// TwinCAT 3 PLC project Mcc
// ProgramVersion: 3.1.4024.0
// libraries:
//   Tc2_Standard, * (Beckhoff Automation GmbH)
//   Tc2_System, * (Beckhoff Automation GmbH)
//   Tc3_Module, * (Beckhoff Automation GmbH)
// project tree:
//   DUTs/ ST_WorkTime.TcDUT
//   POUs/Devices/ Button_NO.TcPOU, Label.TcPOU, Led.TcPOU, MccMotor.TcPOU, MotorContactor.TcPOU, MotorTermFuse.TcPOU, TaurusLed.TcPOU, WorkCounter.TcPOU
//   POUs/Devices/ITFs/ I_Button.TcIO, I_Label.TcIO, I_TaurusLed.TcIO, I_TermFuse.TcIO
//   POUs/ MAIN.TcPOU
// real-time tasks:
//   TASK PlcTask2: cycle T#10ms, priority 22, ADS port 352
// I/O:
//   DEVICE Device 1 (EtherCAT), AmsNetId 192.168.0.130.2.1
//     Term 1 (EK1200) [EK1200-5000 EtherCAT Power supply (2A E-Bus)]
//       Term 2 (EL2008) [EL2008 8Ch. Dig. Output 24V, 0.5A]
//       Term 3 (EL6022) [EL6022 Interface 2Ch. (RS422/485)]
//       Term 4 (EL9011) [EL9011 End Terminal]
//   DEVICE Device 3 (NOV-DP-RAM)
// variable links:
//   MotorControl Instance <-> Device 1 (EtherCAT)/Term 1 (EK1200)/Term 10 (EL2008)
//     PlcTask Outputs/Fermentation_001.MccRev_001.bContactor <-> Channel 1/Fermentation_001.MccRev_001.bContactor
//     PlcTask Outputs/Fermentation_001.MccRev_002.bContactor <-> Channel 2/Fermentation_001.MccRev_002.bContactor
//     PlcTask Outputs/Fermentation_001.MccRev_003.bContactor <-> Channel 3/Fermentation_001.MccRev_003.bContactor
//     PlcTask Outputs/Fermentation_001.MccRev_004.bContactor <-> Channel 4/Fermentation_001.MccRev_004.bContactor
//     PlcTask Outputs/Fermentation_001.MccRev_005.bContactor <-> Channel 5/Fermentation_001.MccRev_005.bContactor
//     PlcTask Outputs/Fermentation_001.MccRev_006.bContactor <-> Channel 6/Fermentation_001.MccRev_006.bContactor
//     PlcTask Outputs/Fermentation_001.MccRev_007.bContactor <-> Channel 7/Fermentation_001.MccRev_007.bContactor
//     PlcTask Outputs/Fermentation_001.MccRev_008.bContactor <-> Channel 8/Fermentation_001.MccRev_008.bContactor
//   MotorControl Instance <-> Device 1 (EtherCAT)/Term 1 (EK1200)/Term 11 (EL2008)
//     PlcTask Outputs/Fermentation_001.MccRev_009.bContactor <-> Channel 1/Fermentation_001.MccRev_009.bContactor
//     PlcTask Outputs/Fermentation_001.MccRev_010.bContactor <-> Channel 2/Fermentation_001.MccRev_010.bContactor
//     PlcTask Outputs/Fermentation_001.MccRev_011.bContactor <-> Channel 3/Fermentation_001.MccRev_011.bContactor
//     PlcTask Outputs/Fermentation_001.MccRev_012.bContactor <-> Channel 4/Fermentation_001.MccRev_012.bContactor
//     PlcTask Outputs/Fermentation_001.MccRev_013.bContactor <-> Channel 5/Fermentation_001.MccRev_013.bContactor
//     PlcTask Outputs/Fermentation_001.MccRev_014.bContactor <-> Channel 6/Fermentation_001.MccRev_014.bContactor
//     PlcTask Outputs/Fermentation_001.MccRev_015.bContactor <-> Channel 7/Fermentation_001.MccRev_015.bContactor
//     PlcTask Outputs/Fermentation_001.MccRev_016.bContactor <-> Channel 8/Fermentation_001.MccRev_016.bContactor
//   MotorControl Instance <-> Device 1 (EtherCAT)/Term 1 (EK1200)/Term 14 (EL3058)
//     PlcTask Inputs/Fermentation_001.TempSens_001.rRawTempValue <-> AI Standard Channel 1/Fermentation_001.TempSens_001.rRawTempValue
//   MotorControl Instance <-> Device 1 (EtherCAT)/Term 1 (EK1200)/Term 2 (EL2008)
//     PlcTask Outputs/Fermentation_001.MccRev_017.bContactor <-> Channel 1/Fermentation_001.MccRev_017.bContactor
//     PlcTask Outputs/Fermentation_001.MccRev_018.bContactor <-> Channel 2/Fermentation_001.MccRev_018.bContactor
//     PlcTask Outputs/Fermentation_001.MccRev_019.bContactor <-> Channel 3/Fermentation_001.MccRev_019.bContactor
//     PlcTask Outputs/Fermentation_001.MccRev_020.bContactor <-> Channel 4/Fermentation_001.MccRev_020.bContactor
//   MotorControl Instance <-> Device 1 (EtherCAT)/Term 1 (EK1200)/Term 6 (EL1008)
//     PlcTask Inputs/Fermentation_001.MccRev_001.bTermFuse <-> Channel 1/Fermentation_001.MccRev_001.bTermFuse
//     PlcTask Inputs/Fermentation_001.MccRev_002.bTermFuse <-> Channel 2/Fermentation_001.MccRev_002.bTermFuse
//     PlcTask Inputs/Fermentation_001.MccRev_003.bTermFuse <-> Channel 3/Fermentation_001.MccRev_003.bTermFuse
//     PlcTask Inputs/Fermentation_001.MccRev_004.bTermFuse <-> Channel 4/Fermentation_001.MccRev_004.bTermFuse
//     PlcTask Inputs/Fermentation_001.MccRev_005.bTermFuse <-> Channel 5/Fermentation_001.MccRev_005.bTermFuse
//     PlcTask Inputs/Fermentation_001.MccRev_006.bTermFuse <-> Channel 6/Fermentation_001.MccRev_006.bTermFuse
//     PlcTask Inputs/Fermentation_001.MccRev_007.bTermFuse <-> Channel 7/Fermentation_001.MccRev_007.bTermFuse
//     PlcTask Inputs/Fermentation_001.MccRev_008.bTermFuse <-> Channel 8/Fermentation_001.MccRev_008.bTermFuse
//   MotorControl Instance <-> Device 1 (EtherCAT)/Term 1 (EK1200)/Term 7 (EL1008)
//     PlcTask Inputs/Fermentation_001.MccRev_009.bTermFuse <-> Channel 1/Fermentation_001.MccRev_009.bTermFuse
//     PlcTask Inputs/Fermentation_001.MccRev_010.bTermFuse <-> Channel 2/Fermentation_001.MccRev_010.bTermFuse
//     PlcTask Inputs/Fermentation_001.MccRev_011.bTermFuse <-> Channel 3/Fermentation_001.MccRev_011.bTermFuse
//     PlcTask Inputs/Fermentation_001.MccRev_012.bTermFuse <-> Channel 4/Fermentation_001.MccRev_012.bTermFuse
//     PlcTask Inputs/Fermentation_001.MccRev_013.bTermFuse <-> Channel 5/Fermentation_001.MccRev_013.bTermFuse
//     PlcTask Inputs/Fermentation_001.MccRev_014.bTermFuse <-> Channel 6/Fermentation_001.MccRev_014.bTermFuse
//     PlcTask Inputs/Fermentation_001.MccRev_015.bTermFuse <-> Channel 7/Fermentation_001.MccRev_015.bTermFuse
//     PlcTask Inputs/Fermentation_001.MccRev_016.bTermFuse <-> Channel 8/Fermentation_001.MccRev_016.bTermFuse
//   MotorControl Instance <-> Device 1 (EtherCAT)/Term 1 (EK1200)/Term 8 (EL1008)
//     PlcTask Inputs/Fermentation_001.MccRev_017.bTermFuse <-> Channel 1/Fermentation_001.MccRev_017.bTermFuse
//     PlcTask Inputs/Fermentation_001.MccRev_018.bTermFuse <-> Channel 2/Fermentation_001.MccRev_018.bTermFuse
//     PlcTask Inputs/Fermentation_001.MccRev_019.bTermFuse <-> Channel 3/Fermentation_001.MccRev_019.bTermFuse
//     PlcTask Inputs/Fermentation_001.MccRev_020.bTermFuse <-> Channel 4/Fermentation_001.MccRev_020.bTermFuse

// ---- DUTs/ST_WorkTime.TcDUT
TYPE ST_WorkTime :
STRUCT
	hours	: UDINT;
	minuts	: UINT;
	seconds	: UINT;
END_STRUCT
END_TYPE

// ---- POUs/Devices/ITFs/I_Button.TcIO
INTERFACE I_Button

PROPERTY IsPressed : BOOL
GET
END_GET
END_PROPERTY

END_INTERFACE

// ---- POUs/Devices/ITFs/I_Label.TcIO
INTERFACE I_Label

PROPERTY Text : STRING
GET
END_GET
SET
END_SET
END_PROPERTY

END_INTERFACE

// ---- POUs/Devices/ITFs/I_TaurusLed.TcIO
INTERFACE I_TaurusLed

PROPERTY Text : STRING
GET
END_GET
SET
END_SET
END_PROPERTY

END_INTERFACE

// ---- POUs/Devices/ITFs/I_TermFuse.TcIO
INTERFACE I_TermFuse

PROPERTY IsActive : BOOL
GET
END_GET
END_PROPERTY

END_INTERFACE

// ---- POUs/Devices/Button_NO.TcPOU
FUNCTION_BLOCK Button_NO IMPLEMENTS I_Button
VAR
	_input AT%M*	:BOOL;
END_VAR

PROPERTY IsPressed : BOOL
GET
IsPressed:= _input;
END_GET
END_PROPERTY

END_FUNCTION_BLOCK

// ---- POUs/Devices/Label.TcPOU
FUNCTION_BLOCK Label IMPLEMENTS I_Label
VAR
	_label AT%M* : T_MaxString;
END_VAR

PROPERTY Text : STRING
GET
Text := _label;
END_GET
SET
_label := Text;
END_SET
END_PROPERTY

END_FUNCTION_BLOCK

// ---- POUs/Devices/Led.TcPOU
FUNCTION_BLOCK Led
VAR
	_state	AT%M* : BOOL;
END_VAR

PROPERTY State : BOOL
GET
State := _state;
END_GET
SET
_state := State;
END_SET
END_PROPERTY

END_FUNCTION_BLOCK

// ---- POUs/Devices/MccMotor.TcPOU
FUNCTION_BLOCK MccMotor
VAR_INPUT
END_VAR
VAR_OUTPUT
END_VAR
VAR
	stWorkTime 				: ST_WorkTime;	// Work time structure
	autoScadaLed			: Led;		// SCADA Led indicated mode of work Mcc
	supplyScadaLed			: Led;		// SCADA Led supply displayed in SCADA it set flag in Memory to read by SCADA
	statusScadaLabel		: Label;	// SCADA Label to display status of Mcc
	workTimeScadaLabel		: Label; 	// SCADA Label to display work time of Mcc 
	autoScadaButton			: Button_NO;		// SCADA Button to set Auto work mode
	forwardScadaButton		: Button_NO;		// SCADA Button to set work Mcc forward
	//reverseScadaButton		: Button_NO;
	stateTaurusLed			: TaurusLed(forwardScadaButton, motorTermFuse, statusScadalabel);	// SCADA Taurus LED to indicate state of Mcc
	motorContactor 			: MotorContactor;	// Psyhical output Starting Contactor 
	motorTermFuse			: MotorTermFuse;	// Psyhical input Thermal and Overcurrent Switch
	motorWorkCounter 		: WorkCounter;	//FB to determine work time of Mcc
	
END_VAR

// Determine the state of the Mcc device
stateTaurusLed();

// Check if MCC is runnning and start count time of work
motorWorkCounter.CheckState(stateTaurusLed);
motorWorkCounter();
motorWorkCounter.MakeString(workTimeScadaLabel);

// Set the supply Led in SCADA system depending on the TermFuse
IF motorTermFuse.IsActive THEN
	supplyScadaLed.State := TRUE;
ELSE
	supplyScadaLed.State := FALSE;
END_IF

// Set the autoScadaLed in SCADA system depending on the AutoScadaButton state
IF autoScadaButton.IsPressed THEN
	autoScadaLed.State := TRUE;
ELSE
	autoScadaLed.State := FALSE;
END_IF

//Logic of Mcc work
IF forwardScadaButton.IsPressed AND motorTermFuse.IsActive THEN
	motorContactor.SwitchOn();
ELSE
	motorContactor.SwitchOff();
END_IF

//Auto/Manual Led set
IF autoScadaButton.IsPressed  THEN
	autoScadaLed.State := TRUE;
ELSE
	autoScadaLed.State := FALSE;
END_IF

END_FUNCTION_BLOCK

// ---- POUs/Devices/TaurusLed.TcPOU
FUNCTION_BLOCK TaurusLed IMPLEMENTS I_TaurusLed
VAR
	_text AT%M* 		: T_MaxString;

	forwardButton		: I_Button;
	motorTermFuse		: I_TermFuse;
	statusScadaLabel	: I_Label;
	
END_VAR

// ustaw stan zmiennej LED Taurusa w TANGO SCADA


statusScadaLabel.Text := 'ON';	

IF motorTermFuse.IsActive THEN
		_text := 'ON';
		statusScadaLabel.Text := 'ON';	
	IF forwardButton.IsPressed THEN
		_text := 'RUNNING';
		statusScadaLabel.Text := 'RUNNING';
	END_IF
ELSE
		_text := 'OFF';
		statusScadaLabel.Text := 'OFF';
	IF forwardButton.IsPressed THEN
		_text := 'FAULT';
		statusScadaLabel.Text := 'FAULT';
	END_IF
END_IF

METHOD FB_init : BOOL
VAR_INPUT
	bInitRetains 		: BOOL; // if TRUE, the retain variables are initialized (warm start / cold start)
	bInCopyCode 		: BOOL;  // if TRUE, the instance afterwards gets moved into the copy code (online change)
	forwardButton		: I_Button;
	motorTermFuse		: I_TermFuse;
	statusScadaLabel	: I_Label;
END_VAR
THIS^.forwardButton			:= forwardButton;
THIS^.motorTermFuse			:= motorTermFuse;
THIS^.statusScadaLabel      := statusScadaLabel;
END_METHOD

PROPERTY Text : STRING
GET
Text := _text;
END_GET
SET
_text := Text;
END_SET
END_PROPERTY

END_FUNCTION_BLOCK

// ---- POUs/Devices/MotorTermFuse.TcPOU
FUNCTION_BLOCK MotorTermFuse IMPLEMENTS I_TermFuse
VAR
	_input AT%I* :BOOL;
	
END_VAR

PROPERTY IsActive : BOOL
GET
IsActive := _input;
END_GET
END_PROPERTY

END_FUNCTION_BLOCK

// ---- POUs/Devices/MotorContactor.TcPOU
FUNCTION_BLOCK MotorContactor
VAR
	_output	AT%Q*	: BOOL;
END_VAR

METHOD SwitchOff : BOOL
VAR_INPUT
END_VAR
_output := False;
END_METHOD

METHOD SwitchOn : BOOL
VAR_INPUT
END_VAR
_output := True;
END_METHOD

END_FUNCTION_BLOCK

// ---- POUs/Devices/WorkCounter.TcPOU
FUNCTION_BLOCK WorkCounter
VAR
	startCount  : BOOL;
	stWorkTime  : ST_WorkTime;
	fbTon		: TON;
	_text	    : T_MaxString;
	
END_VAR

fbTon(IN := TRUE, PT := T#1S);

IF (fbTon.Q) AND startCount THEN
	
	fbTon(IN:=FALSE);
	stWorkTime.seconds := stWorkTime.seconds +1;
	
	IF stWorkTime.seconds > 59 THEN
		stWorkTime.seconds := 0;
		stWorkTime.minuts := stWorkTime.minuts +1;
		IF stWorkTime.minuts > 59 THEN
			stWorkTime.minuts := 0;
			stWorkTime.hours := stWorkTime.hours +1;	
		END_IF
	END_IF
	
END_IF

METHOD CheckState : BOOL
VAR_INPUT
	iTaurusLed	: I_TaurusLed;
END_VAR
IF iTaurusLed.Text = 'RUNNING' THEN
	THIS^.startCount := TRUE;
ELSE
	THIS^.startCount := FALSE;
END_IF
END_METHOD

METHOD MakeString : STRING
VAR_INPUT
	workTimeScadaLabel	: I_Label;
END_VAR
// Forms a chain of the form 'Hours:Minuts:Seconds'
THIS^._text := CONCAT(UDINT_TO_STRING(THIS^.stWorkTime.hours), ':');
THIS^._text := CONCAT(THIS^._text, UDINT_TO_STRING(THIS^.stWorkTime.minuts));
THIS^._text := CONCAT(THIS^._text, ':');
THIS^._text := CONCAT(THIS^._text, UDINT_TO_STRING(stWorkTime.seconds));

workTimeScadaLabel.Text := THIS^._text;
END_METHOD

END_FUNCTION_BLOCK

// ---- POUs/MAIN.TcPOU
PROGRAM MAIN
VAR
	
	mccMotor				: MccMotor;
	mccMotorP01				: MccMotor;

//	stWorkTime 				: ST_WorkTime;
//	autoScadaLed			: Led;
//	supplyScadaLed			: Led;
//	statusScadaLabel		: Label;
//	motorContactor 			: MotorContactor;
//	motorTermFuse			: MotorTermFuse;
//	autoScadaButton			: Button_NO;
//	forwardScadaButton		: Button_NO;
//	reverseScadaButton		: Button_NO;
//	stateTaurusLed			: TaurusLed(forwardScadaButton, motorTermFuse);
//	motorWorkTime 			: WorkCounter;
	
	
	
END_VAR

;
//mccMotor();
//mccMotorP01();

END_PROGRAM
